(* Logix 5000 project; controller CarbonScout_MK6 vendor 1 type 14 code 154 rev 32.11; software revision 32.00; part 14 of 17 *)
(* tags used below, declared in another part *)
   i : DINT;
   Index : DINT;
   LocalSampleTank : DINT;
   LOnlineNumber : DINT;
   ManualRunning : BOOL;
   ONS : BOOL[32];
   TimeRemainingCal : TimeRemainingCal;
   AI_LIT_02 : P_AIn;   // Carbon Scout Cone Level Transmitter
   CS_DINTParams : DINT[100];
   CS_REALParams : REAL[80];   // CS REAL Parameters
   CS_ResultStore : CS_Results[20,20];   // Sample Result Historical
   CS_Seq : GEK_Sequence;
   CS_Tank : CS_TankParams[20];
   CS_Timer : TIMER[80];
   Reg_Cal : REAL[10];   // working calculation variables
   Reg_Calsum : REAL[10];   // running sum of calc variables
   Reg_DINTparams : DINT[8];   // Dint and bools for calcs
   Reg_InX : REAL[30];   // X input for calcs
   Reg_InY : REAL[30];   // Y input for pairs
   Reg_Model : REAL[4];   // Calculated model output and site model
   Reg_Out : REAL[14];   // Output of calculation
   TimeAndDate : DINT[7];
   Valve_XV_15 : P_ValveSO;   // Bottme wash vavle
(* SeqProgram, continued *)

ROUTINE DataShift   (* ladder *)
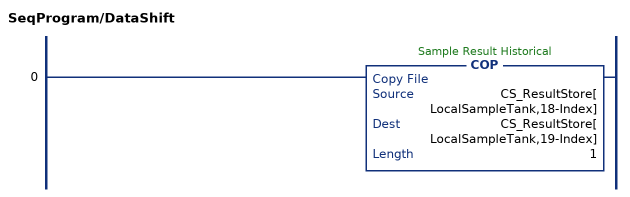
   0: COP(CS_ResultStore[LocalSampleTank,18-Index],CS_ResultStore[LocalSampleTank,19-Index],1);
END_ROUTINE

ROUTINE MainRoutine   (* ladder *)
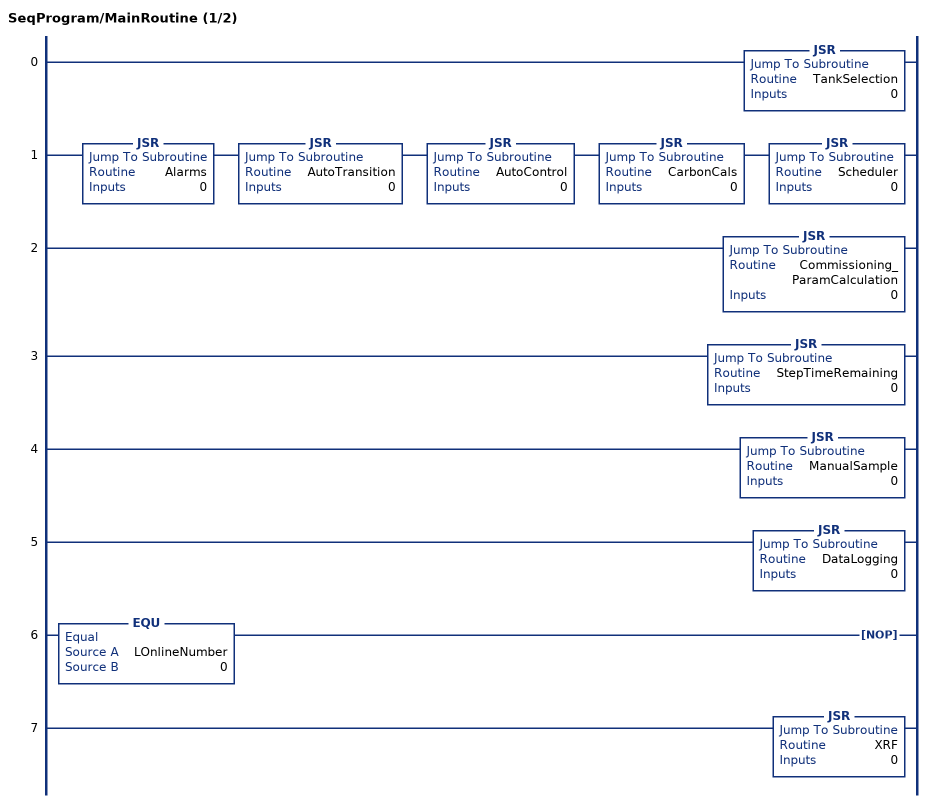
   0: JSR(TankSelection,0);
   1: JSR(Alarms,0)JSR(AutoTransition,0)JSR(AutoControl,0)JSR(CarbonCals,0)JSR(Scheduler,0);
   2: JSR(Commissioning_ParamCalculation,0);
   3: JSR(StepTimeRemaining,0);
   4: JSR(ManualSample,0);
   5: JSR(DataLogging,0);
   6: EQU(LOnlineNumber,0)NOP();
   7: JSR(XRF,0);
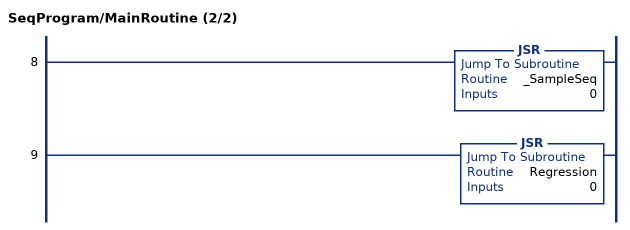
   8: JSR(_SampleSeq,0);
   9: JSR(Regression,0);
END_ROUTINE

ROUTINE ManualSample   (* ladder *)
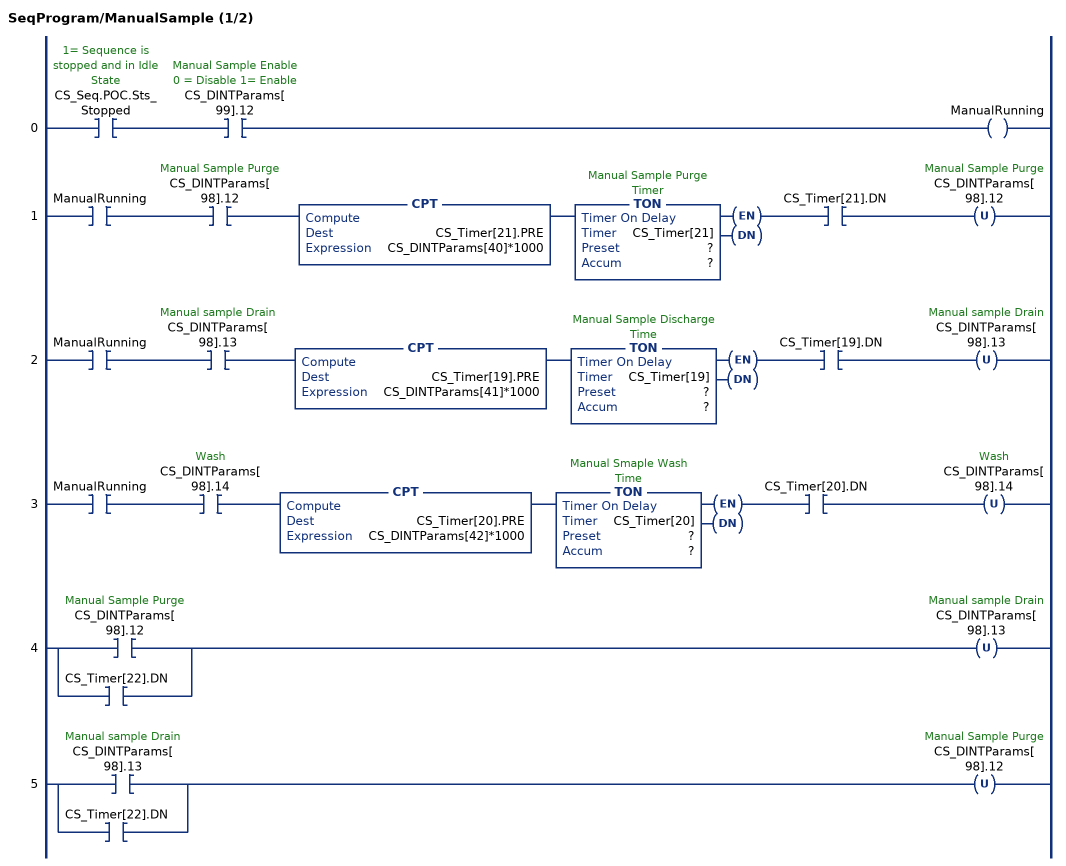
   0: XIC(CS_Seq.POC.Sts_Stopped)XIC(CS_DINTParams[99].12)OTE(ManualRunning);
   1: XIC(ManualRunning)XIC(CS_DINTParams[98].12)CPT(CS_Timer[21].PRE,CS_DINTParams[40]*1000)TON(CS_Timer[21],?,?)XIC(CS_Timer[21].DN)OTU(CS_DINTParams[98].12);
   2: XIC(ManualRunning)XIC(CS_DINTParams[98].13)CPT(CS_Timer[19].PRE,CS_DINTParams[41]*1000)TON(CS_Timer[19],?,?)XIC(CS_Timer[19].DN)OTU(CS_DINTParams[98].13);
   3: XIC(ManualRunning)XIC(CS_DINTParams[98].14)CPT(CS_Timer[20].PRE,CS_DINTParams[42]*1000)TON(CS_Timer[20],?,?)XIC(CS_Timer[20].DN)OTU(CS_DINTParams[98].14);
   4: [XIC(CS_DINTParams[98].12) ,XIC(CS_Timer[22].DN) ]OTU(CS_DINTParams[98].13);
   5: [XIC(CS_DINTParams[98].13) ,XIC(CS_Timer[22].DN) ]OTU(CS_DINTParams[98].12);
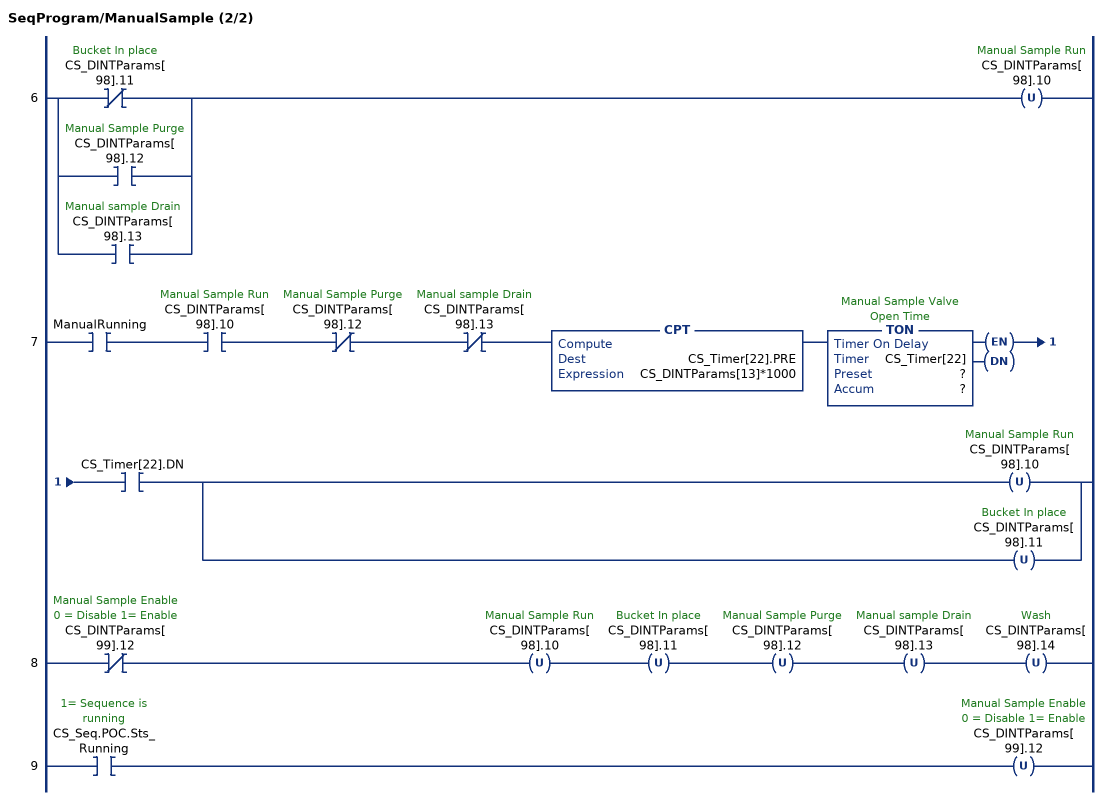
   6: [XIO(CS_DINTParams[98].11) ,XIC(CS_DINTParams[98].12) ,XIC(CS_DINTParams[98].13) ]OTU(CS_DINTParams[98].10);
   7: XIC(ManualRunning)XIC(CS_DINTParams[98].10)XIO(CS_DINTParams[98].12)XIO(CS_DINTParams[98].13)CPT(CS_Timer[22].PRE,CS_DINTParams[13]*1000)TON(CS_Timer[22],?,?)XIC(CS_Timer[22].DN)[OTU(CS_DINTParams[98].10) ,OTU(CS_DINTParams[98].11) ];
   8: XIO(CS_DINTParams[99].12)OTU(CS_DINTParams[98].10)OTU(CS_DINTParams[98].11)OTU(CS_DINTParams[98].12)OTU(CS_DINTParams[98].13)OTU(CS_DINTParams[98].14);
   9: XIC(CS_Seq.POC.Sts_Running)OTU(CS_DINTParams[99].12);
END_ROUTINE

ROUTINE Regression   (* ladder *)
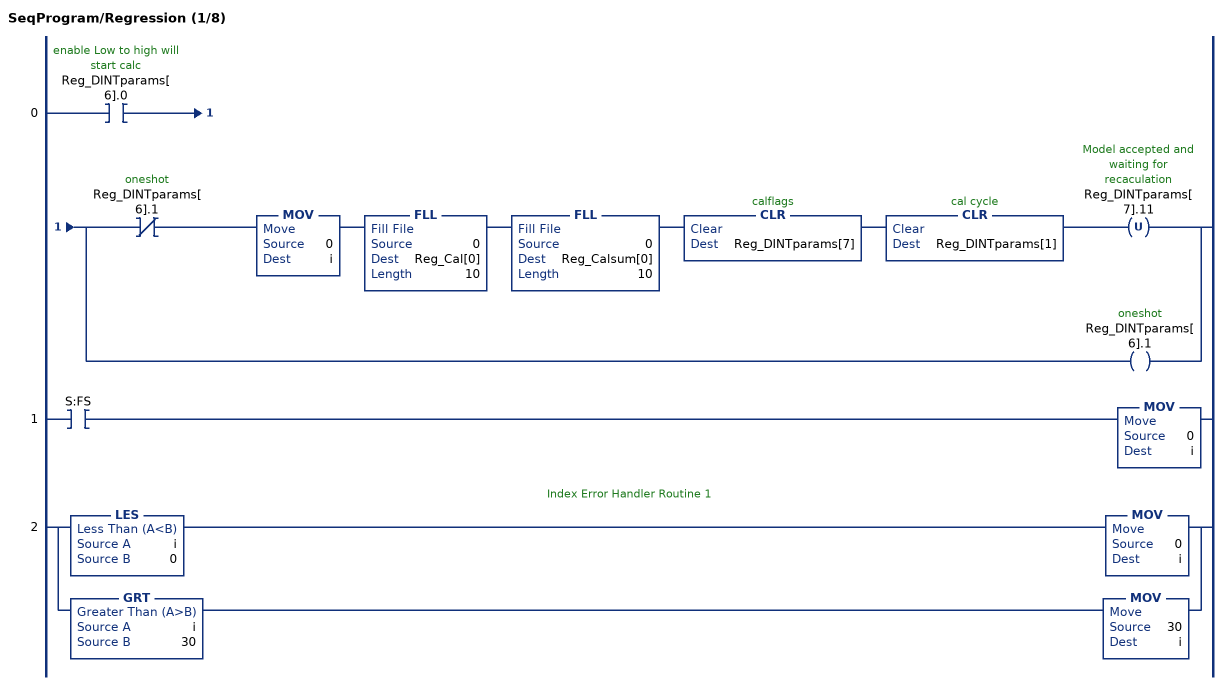
   0: XIC(Reg_DINTparams[6].0)[XIO(Reg_DINTparams[6].1) MOV(0,i) FLL(0,Reg_Cal[0],10) FLL(0,Reg_Calsum[0],10) CLR(Reg_DINTparams[7]) CLR(Reg_DINTparams[1]) OTU(Reg_DINTparams[7].11) ,OTE(Reg_DINTparams[6].1) ];
   1: XIC(S:FS)MOV(0,i);
   // Index Error Handler Routine 1
   2: [LES(i,0) MOV(0,i) ,GRT(i,30) MOV(30,i) ];
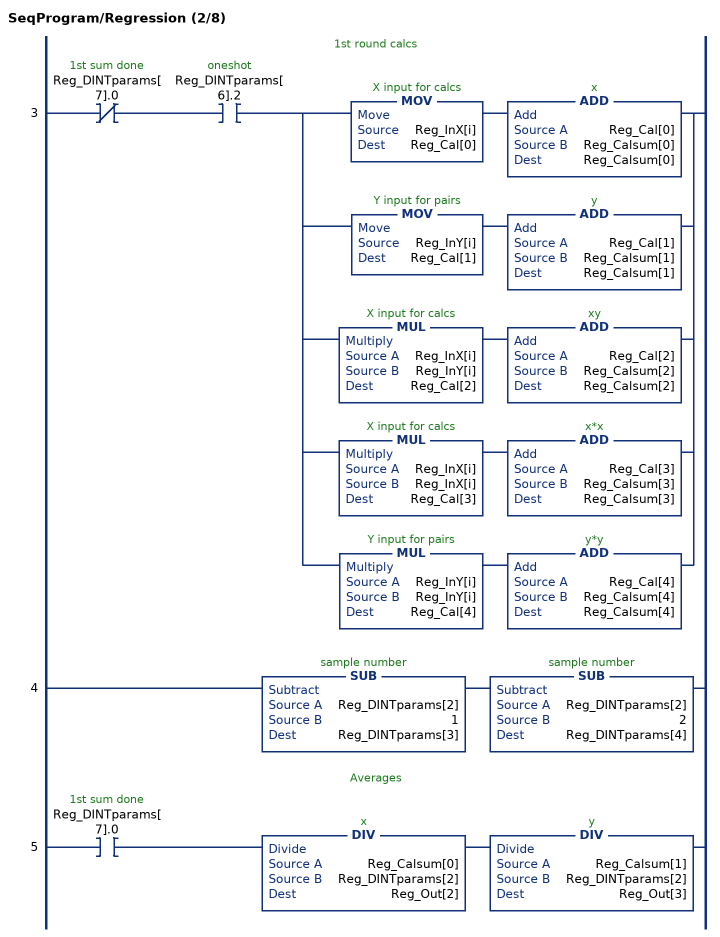
   // 1st round calcs
   3: XIO(Reg_DINTparams[7].0)XIC(Reg_DINTparams[6].2)[MOV(Reg_InX[i],Reg_Cal[0]) ADD(Reg_Cal[0],Reg_Calsum[0],Reg_Calsum[0]) ,MOV(Reg_InY[i],Reg_Cal[1]) ADD(Reg_Cal[1],Reg_Calsum[1],Reg_Calsum[1]) ,MUL(Reg_InX[i],Reg_InY[i],Reg_Cal[2]) ADD(Reg_Cal[2],Reg_Calsum[2],Reg_Calsum[2]) ,MUL(Reg_InX[i],Reg_InX[i],Reg_Cal[3]) ADD(Reg_Cal[3],Reg_Calsum[3],Reg_Calsum[3]) ,MUL(Reg_InY[i],Reg_InY[i],Reg_Cal[4]) ADD(Reg_Cal[4],Reg_Calsum[4],Reg_Calsum[4]) ];
   4: SUB(Reg_DINTparams[2],1,Reg_DINTparams[3])SUB(Reg_DINTparams[2],2,Reg_DINTparams[4]);
   // Averages
   5: XIC(Reg_DINTparams[7].0)DIV(Reg_Calsum[0],Reg_DINTparams[2],Reg_Out[2])DIV(Reg_Calsum[1],Reg_DINTparams[2],Reg_Out[3]);
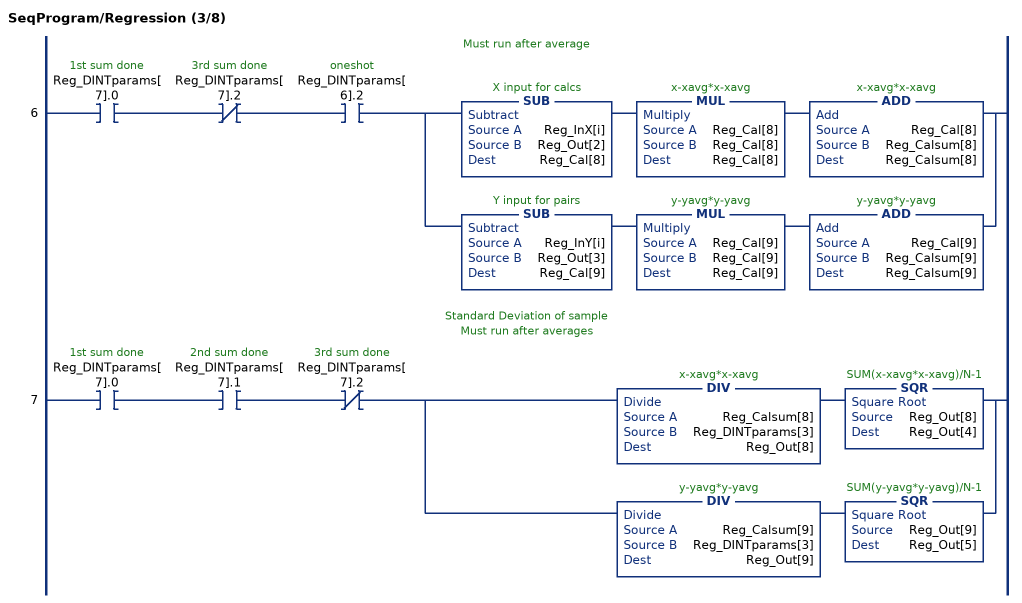
   // Must run after average
   6: XIC(Reg_DINTparams[7].0)XIO(Reg_DINTparams[7].2)XIC(Reg_DINTparams[6].2)[SUB(Reg_InX[i],Reg_Out[2],Reg_Cal[8]) MUL(Reg_Cal[8],Reg_Cal[8],Reg_Cal[8]) ADD(Reg_Cal[8],Reg_Calsum[8],Reg_Calsum[8]) ,SUB(Reg_InY[i],Reg_Out[3],Reg_Cal[9]) MUL(Reg_Cal[9],Reg_Cal[9],Reg_Cal[9]) ADD(Reg_Cal[9],Reg_Calsum[9],Reg_Calsum[9]) ];
   // Standard Deviation of sample
   // Must run after averages
   7: XIC(Reg_DINTparams[7].0)XIC(Reg_DINTparams[7].1)XIO(Reg_DINTparams[7].2)[DIV(Reg_Calsum[8],Reg_DINTparams[3],Reg_Out[8]) SQR(Reg_Out[8],Reg_Out[4]) ,DIV(Reg_Calsum[9],Reg_DINTparams[3],Reg_Out[9]) SQR(Reg_Out[9],Reg_Out[5]) ];
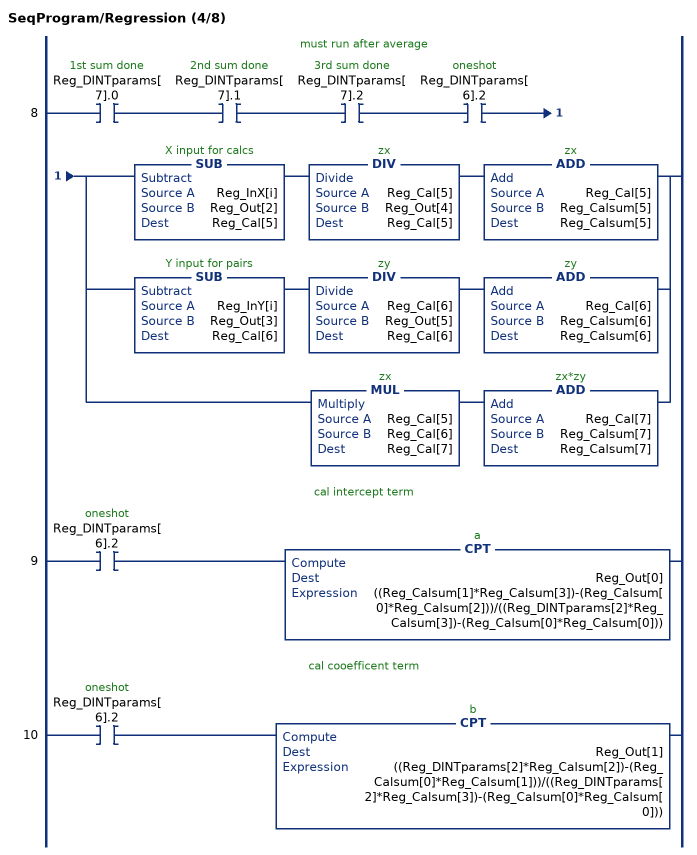
   // must run after average
   8: XIC(Reg_DINTparams[7].0)XIC(Reg_DINTparams[7].1)XIC(Reg_DINTparams[7].2)XIC(Reg_DINTparams[6].2)[SUB(Reg_InX[i],Reg_Out[2],Reg_Cal[5]) DIV(Reg_Cal[5],Reg_Out[4],Reg_Cal[5]) ADD(Reg_Cal[5],Reg_Calsum[5],Reg_Calsum[5]) ,SUB(Reg_InY[i],Reg_Out[3],Reg_Cal[6]) DIV(Reg_Cal[6],Reg_Out[5],Reg_Cal[6]) ADD(Reg_Cal[6],Reg_Calsum[6],Reg_Calsum[6]) ,MUL(Reg_Cal[5],Reg_Cal[6],Reg_Cal[7]) ADD(Reg_Cal[7],Reg_Calsum[7],Reg_Calsum[7]) ];
   // cal intercept term
   9: XIC(Reg_DINTparams[6].2)CPT(Reg_Out[0],((Reg_Calsum[1]*Reg_Calsum[3])-(Reg_Calsum[0]*Reg_Calsum[2]))/((Reg_DINTparams[2]*Reg_Calsum[3])-(Reg_Calsum[0]*Reg_Calsum[0])));
   // cal cooefficent term
   10: XIC(Reg_DINTparams[6].2)CPT(Reg_Out[1],((Reg_DINTparams[2]*Reg_Calsum[2])-(Reg_Calsum[0]*Reg_Calsum[1]))/((Reg_DINTparams[2]*Reg_Calsum[3])-(Reg_Calsum[0]*Reg_Calsum[0])));
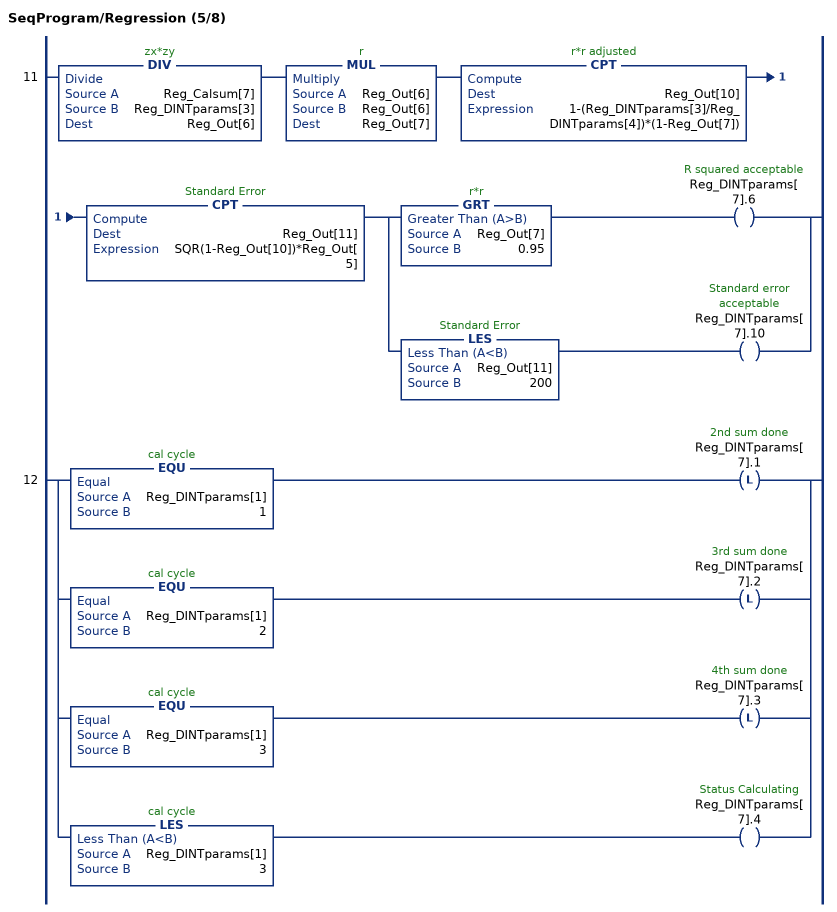
   11: DIV(Reg_Calsum[7],Reg_DINTparams[3],Reg_Out[6])MUL(Reg_Out[6],Reg_Out[6],Reg_Out[7])CPT(Reg_Out[10],1-(Reg_DINTparams[3]/Reg_DINTparams[4])*(1-Reg_Out[7]))CPT(Reg_Out[11],SQR(1-Reg_Out[10])*Reg_Out[5])[GRT(Reg_Out[7],0.95) OTE(Reg_DINTparams[7].6) ,LES(Reg_Out[11],200) OTE(Reg_DINTparams[7].10) ];
   12: [EQU(Reg_DINTparams[1],1) OTL(Reg_DINTparams[7].1) ,EQU(Reg_DINTparams[1],2) OTL(Reg_DINTparams[7].2) ,EQU(Reg_DINTparams[1],3) OTL(Reg_DINTparams[7].3) ,LES(Reg_DINTparams[1],3) OTE(Reg_DINTparams[7].4) ];
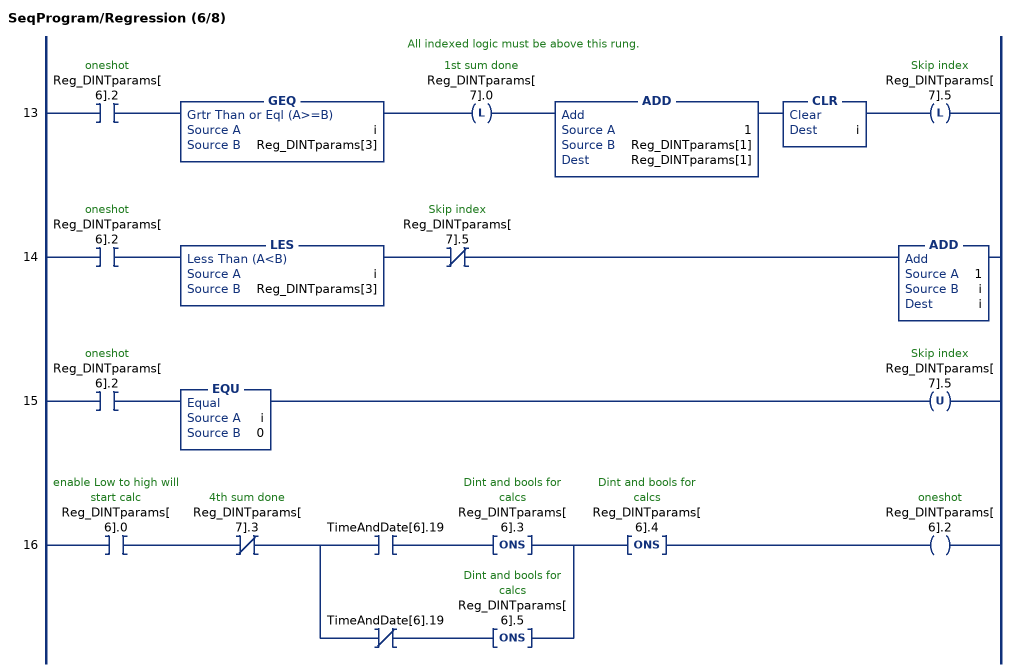
   // All indexed logic must be above this rung.
   13: XIC(Reg_DINTparams[6].2)GEQ(i,Reg_DINTparams[3])OTL(Reg_DINTparams[7].0)ADD(1,Reg_DINTparams[1],Reg_DINTparams[1])CLR(i)OTL(Reg_DINTparams[7].5);
   14: XIC(Reg_DINTparams[6].2)LES(i,Reg_DINTparams[3])XIO(Reg_DINTparams[7].5)ADD(1,i,i);
   15: XIC(Reg_DINTparams[6].2)EQU(i,0)OTU(Reg_DINTparams[7].5);
   16: XIC(Reg_DINTparams[6].0)XIO(Reg_DINTparams[7].3)[XIC(TimeAndDate[6].19) ONS(Reg_DINTparams[6].3) ,XIO(TimeAndDate[6].19) ONS(Reg_DINTparams[6].5) ]ONS(Reg_DINTparams[6].4)OTE(Reg_DINTparams[6].2);
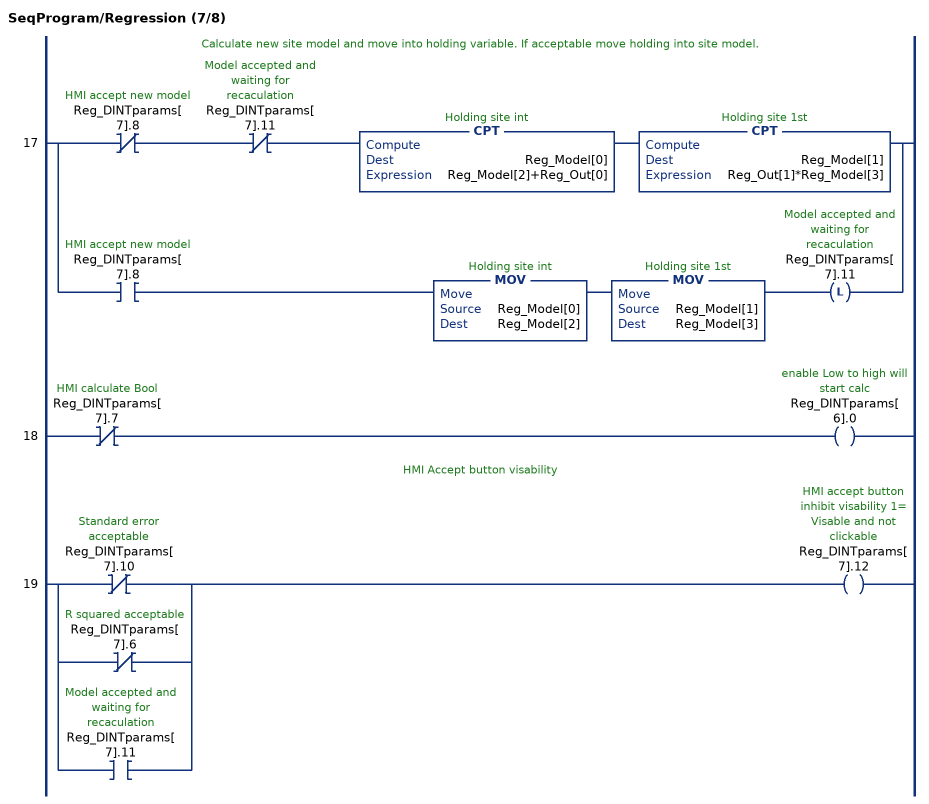
   // Calculate new site model and move into holding variable. If acceptable move holding into site model.
   17: [XIO(Reg_DINTparams[7].8) XIO(Reg_DINTparams[7].11) CPT(Reg_Model[0],Reg_Model[2]+Reg_Out[0]) CPT(Reg_Model[1],Reg_Out[1]*Reg_Model[3]) ,XIC(Reg_DINTparams[7].8) MOV(Reg_Model[0],Reg_Model[2]) MOV(Reg_Model[1],Reg_Model[3]) OTL(Reg_DINTparams[7].11) ];
   18: XIO(Reg_DINTparams[7].7)OTE(Reg_DINTparams[6].0);
   // HMI Accept button visability
   19: [XIO(Reg_DINTparams[7].10) ,XIO(Reg_DINTparams[7].6) ,XIC(Reg_DINTparams[7].11) ]OTE(Reg_DINTparams[7].12);
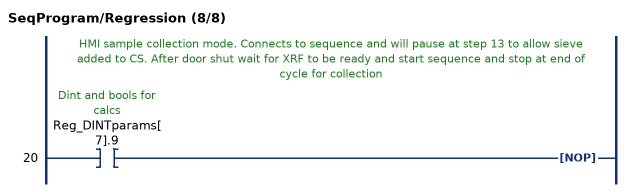
   // HMI sample collection mode. Connects to sequence and will pause at step 13 to allow sieve added to CS. After door shut wait for XRF to be ready and start sequence and stop at end of cycle for collection
   20: XIC(Reg_DINTparams[7].9)NOP();
END_ROUTINE

ROUTINE Scheduler   (* ladder *)
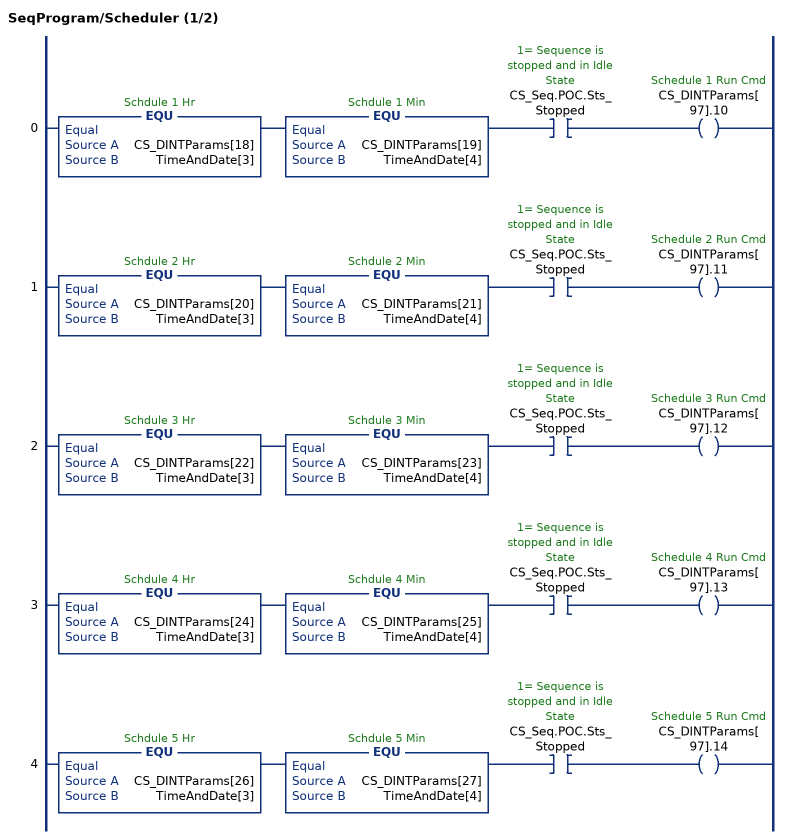
   0: EQU(CS_DINTParams[18],TimeAndDate[3])EQU(CS_DINTParams[19],TimeAndDate[4])XIC(CS_Seq.POC.Sts_Stopped)OTE(CS_DINTParams[97].10);
   1: EQU(CS_DINTParams[20],TimeAndDate[3])EQU(CS_DINTParams[21],TimeAndDate[4])XIC(CS_Seq.POC.Sts_Stopped)OTE(CS_DINTParams[97].11);
   2: EQU(CS_DINTParams[22],TimeAndDate[3])EQU(CS_DINTParams[23],TimeAndDate[4])XIC(CS_Seq.POC.Sts_Stopped)OTE(CS_DINTParams[97].12);
   3: EQU(CS_DINTParams[24],TimeAndDate[3])EQU(CS_DINTParams[25],TimeAndDate[4])XIC(CS_Seq.POC.Sts_Stopped)OTE(CS_DINTParams[97].13);
   4: EQU(CS_DINTParams[26],TimeAndDate[3])EQU(CS_DINTParams[27],TimeAndDate[4])XIC(CS_Seq.POC.Sts_Stopped)OTE(CS_DINTParams[97].14);
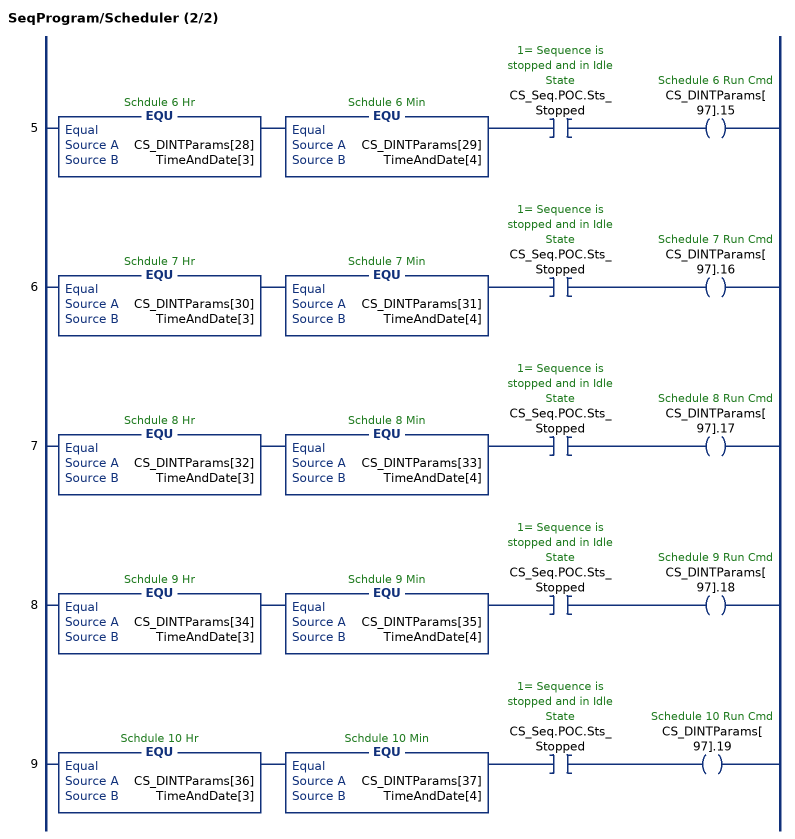
   5: EQU(CS_DINTParams[28],TimeAndDate[3])EQU(CS_DINTParams[29],TimeAndDate[4])XIC(CS_Seq.POC.Sts_Stopped)OTE(CS_DINTParams[97].15);
   6: EQU(CS_DINTParams[30],TimeAndDate[3])EQU(CS_DINTParams[31],TimeAndDate[4])XIC(CS_Seq.POC.Sts_Stopped)OTE(CS_DINTParams[97].16);
   7: EQU(CS_DINTParams[32],TimeAndDate[3])EQU(CS_DINTParams[33],TimeAndDate[4])XIC(CS_Seq.POC.Sts_Stopped)OTE(CS_DINTParams[97].17);
   8: EQU(CS_DINTParams[34],TimeAndDate[3])EQU(CS_DINTParams[35],TimeAndDate[4])XIC(CS_Seq.POC.Sts_Stopped)OTE(CS_DINTParams[97].18);
   9: EQU(CS_DINTParams[36],TimeAndDate[3])EQU(CS_DINTParams[37],TimeAndDate[4])XIC(CS_Seq.POC.Sts_Stopped)OTE(CS_DINTParams[97].19);
END_ROUTINE

ROUTINE StepTimeRemaining   (* ladder *)
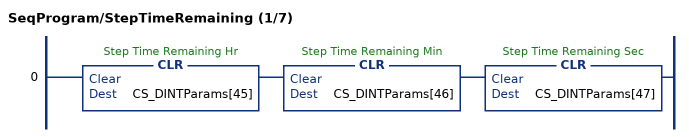
   0: CLR(CS_DINTParams[45])CLR(CS_DINTParams[46])CLR(CS_DINTParams[47]);
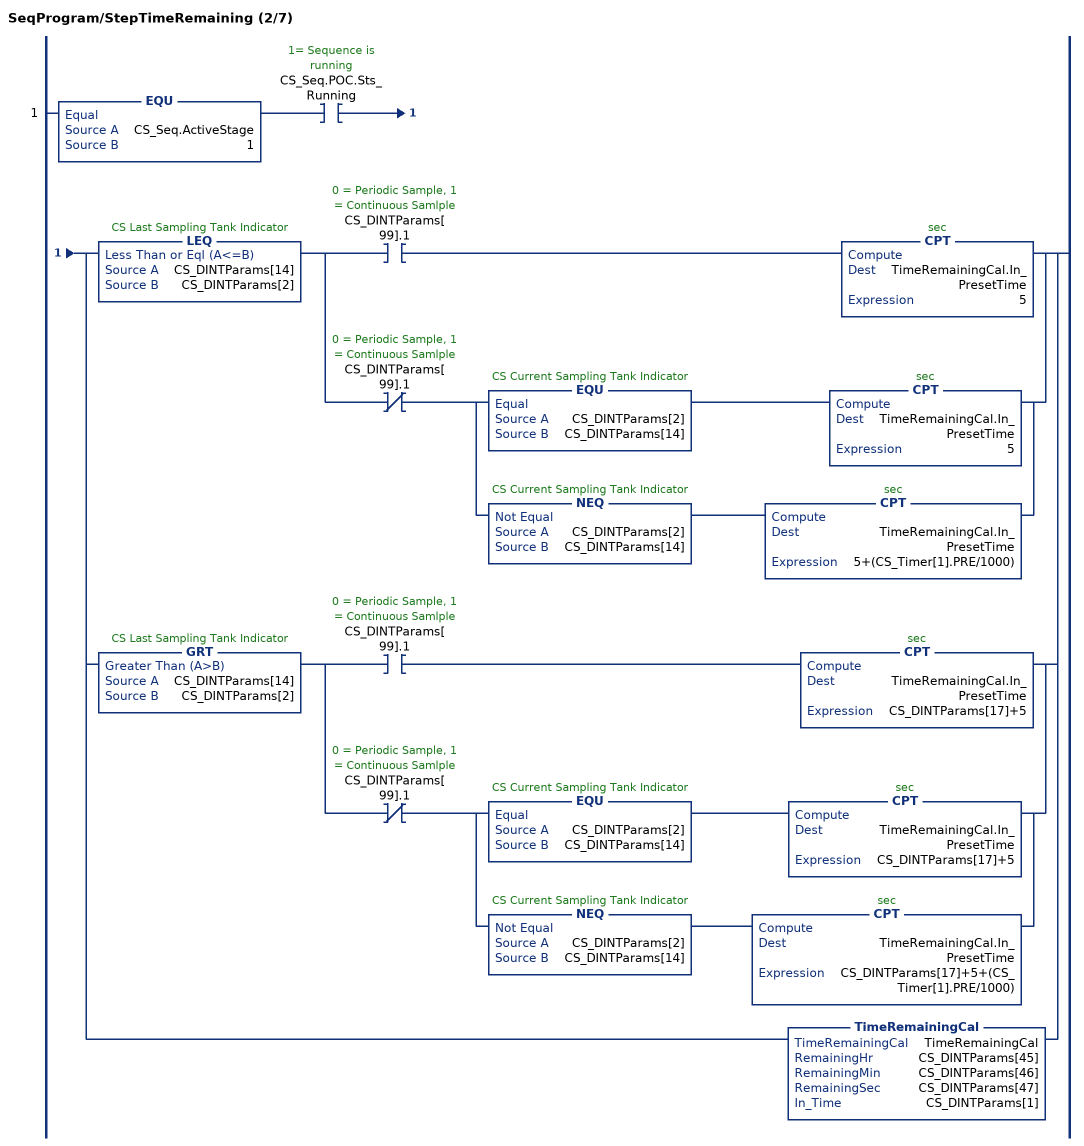
   1: EQU(CS_Seq.ActiveStage,1)XIC(CS_Seq.POC.Sts_Running)[[LEQ(CS_DINTParams[14],CS_DINTParams[2]) [XIC(CS_DINTParams[99].1) CPT(TimeRemainingCal.In_PresetTime,5) ,XIO(CS_DINTParams[99].1) [EQU(CS_DINTParams[2],CS_DINTParams[14]) CPT(TimeRemainingCal.In_PresetTime,5) ,NEQ(CS_DINTParams[2],CS_DINTParams[14]) CPT(TimeRemainingCal.In_PresetTime,5+(CS_Timer[1].PRE/1000)) ] ] ,GRT(CS_DINTParams[14],CS_DINTParams[2]) [XIC(CS_DINTParams[99].1) CPT(TimeRemainingCal.In_PresetTime,CS_DINTParams[17]+5) ,XIO(CS_DINTParams[99].1) [EQU(CS_DINTParams[2],CS_DINTParams[14]) CPT(TimeRemainingCal.In_PresetTime,CS_DINTParams[17]+5) ,NEQ(CS_DINTParams[2],CS_DINTParams[14]) CPT(TimeRemainingCal.In_PresetTime,CS_DINTParams[17]+5+(CS_Timer[1].PRE/1000)) ] ] ] ,TimeRemainingCal(TimeRemainingCal,CS_DINTParams[45],CS_DINTParams[46],CS_DINTParams[47],CS_DINTParams[1]) ];
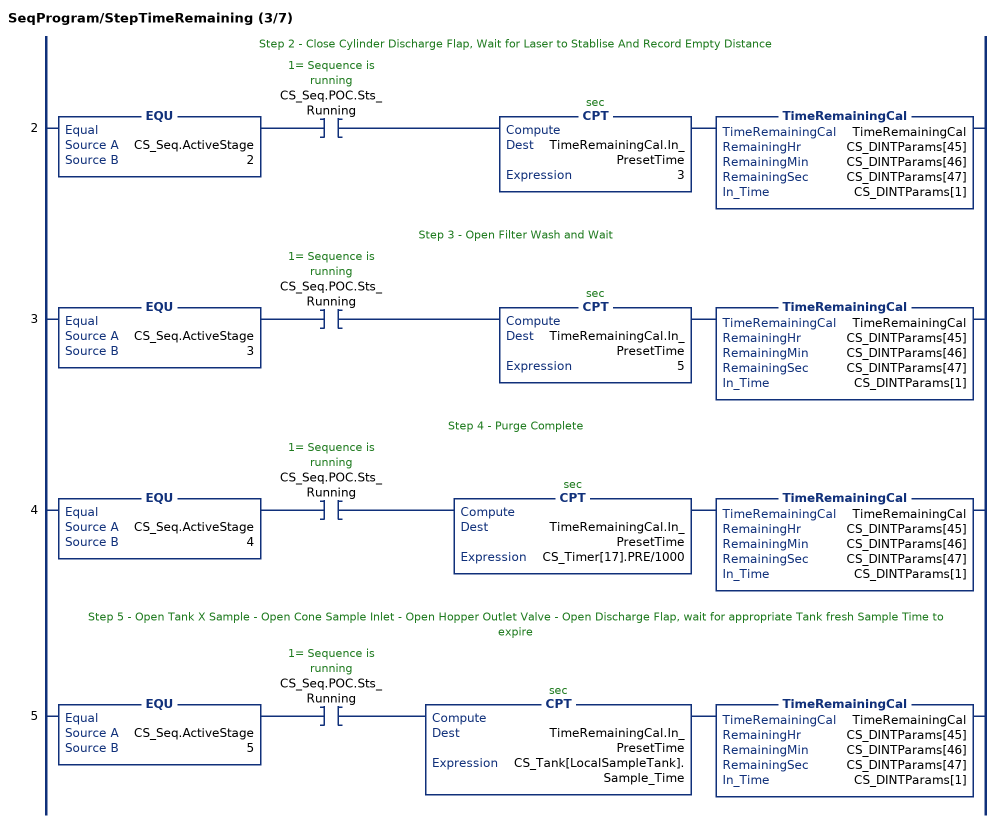
   // Step 2 - Close Cylinder Discharge Flap, Wait for Laser to Stablise And Record Empty Distance
   2: EQU(CS_Seq.ActiveStage,2)XIC(CS_Seq.POC.Sts_Running)CPT(TimeRemainingCal.In_PresetTime,3)TimeRemainingCal(TimeRemainingCal,CS_DINTParams[45],CS_DINTParams[46],CS_DINTParams[47],CS_DINTParams[1]);
   // Step 3 - Open Filter Wash and Wait
   3: EQU(CS_Seq.ActiveStage,3)XIC(CS_Seq.POC.Sts_Running)CPT(TimeRemainingCal.In_PresetTime,5)TimeRemainingCal(TimeRemainingCal,CS_DINTParams[45],CS_DINTParams[46],CS_DINTParams[47],CS_DINTParams[1]);
   // Step 4 - Purge Complete
   4: EQU(CS_Seq.ActiveStage,4)XIC(CS_Seq.POC.Sts_Running)CPT(TimeRemainingCal.In_PresetTime,CS_Timer[17].PRE/1000)TimeRemainingCal(TimeRemainingCal,CS_DINTParams[45],CS_DINTParams[46],CS_DINTParams[47],CS_DINTParams[1]);
   // Step 5 - Open Tank X Sample - Open Cone Sample Inlet - Open Hopper Outlet Valve - Open Discharge Flap, wait for appropriate Tank fresh Sample Time to expire
   5: EQU(CS_Seq.ActiveStage,5)XIC(CS_Seq.POC.Sts_Running)CPT(TimeRemainingCal.In_PresetTime,CS_Tank[LocalSampleTank].Sample_Time)TimeRemainingCal(TimeRemainingCal,CS_DINTParams[45],CS_DINTParams[46],CS_DINTParams[47],CS_DINTParams[1]);
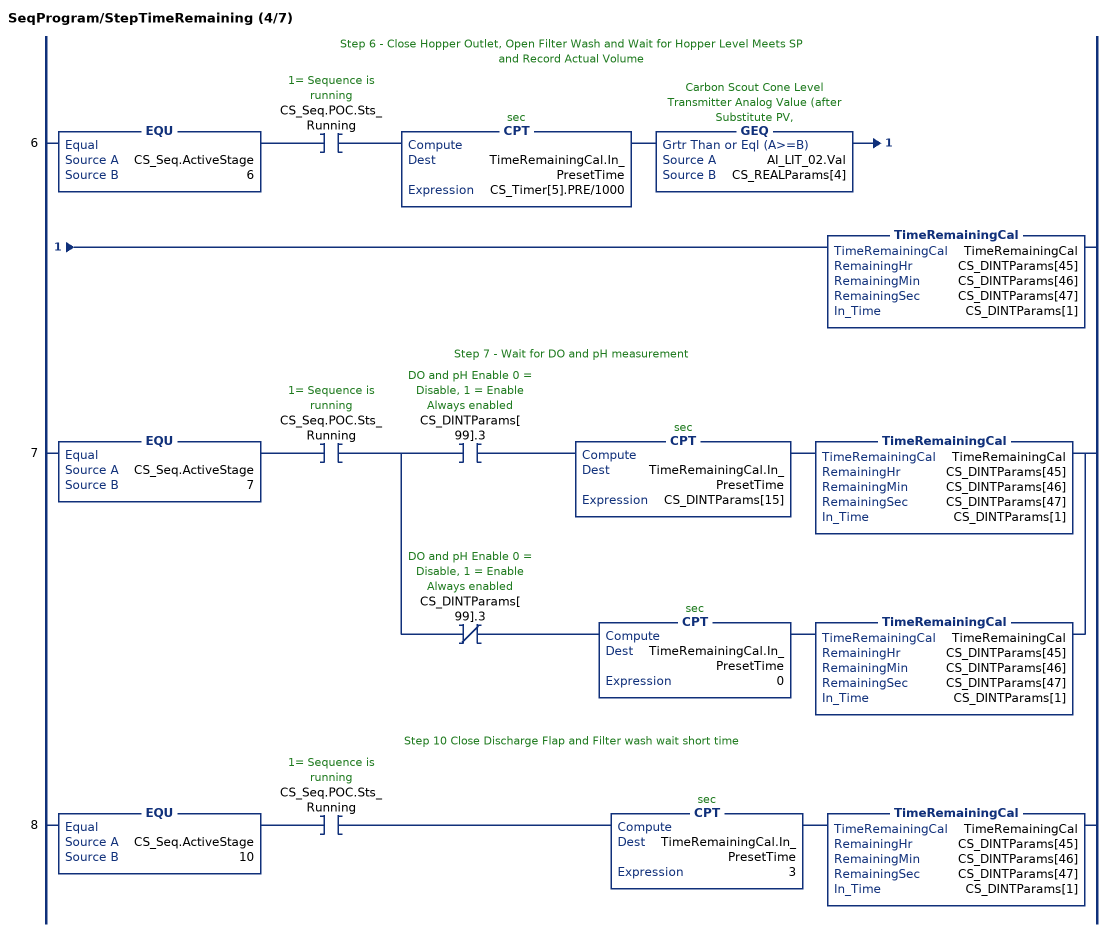
   // Step 6 - Close Hopper Outlet, Open Filter Wash and Wait for Hopper Level Meets SP
   // and Record Actual Volume
   6: EQU(CS_Seq.ActiveStage,6)XIC(CS_Seq.POC.Sts_Running)CPT(TimeRemainingCal.In_PresetTime,CS_Timer[5].PRE/1000)GEQ(AI_LIT_02.Val,CS_REALParams[4])TimeRemainingCal(TimeRemainingCal,CS_DINTParams[45],CS_DINTParams[46],CS_DINTParams[47],CS_DINTParams[1]);
   // Step 7 - Wait for DO and pH measurement
   7: EQU(CS_Seq.ActiveStage,7)XIC(CS_Seq.POC.Sts_Running)[XIC(CS_DINTParams[99].3) CPT(TimeRemainingCal.In_PresetTime,CS_DINTParams[15]) TimeRemainingCal(TimeRemainingCal,CS_DINTParams[45],CS_DINTParams[46],CS_DINTParams[47],CS_DINTParams[1]) ,XIO(CS_DINTParams[99].3) CPT(TimeRemainingCal.In_PresetTime,0) TimeRemainingCal(TimeRemainingCal,CS_DINTParams[45],CS_DINTParams[46],CS_DINTParams[47],CS_DINTParams[1]) ];
   // Step 10 Close Discharge Flap and Filter wash wait short time
   8: EQU(CS_Seq.ActiveStage,10)XIC(CS_Seq.POC.Sts_Running)CPT(TimeRemainingCal.In_PresetTime,3)TimeRemainingCal(TimeRemainingCal,CS_DINTParams[45],CS_DINTParams[46],CS_DINTParams[47],CS_DINTParams[1]);
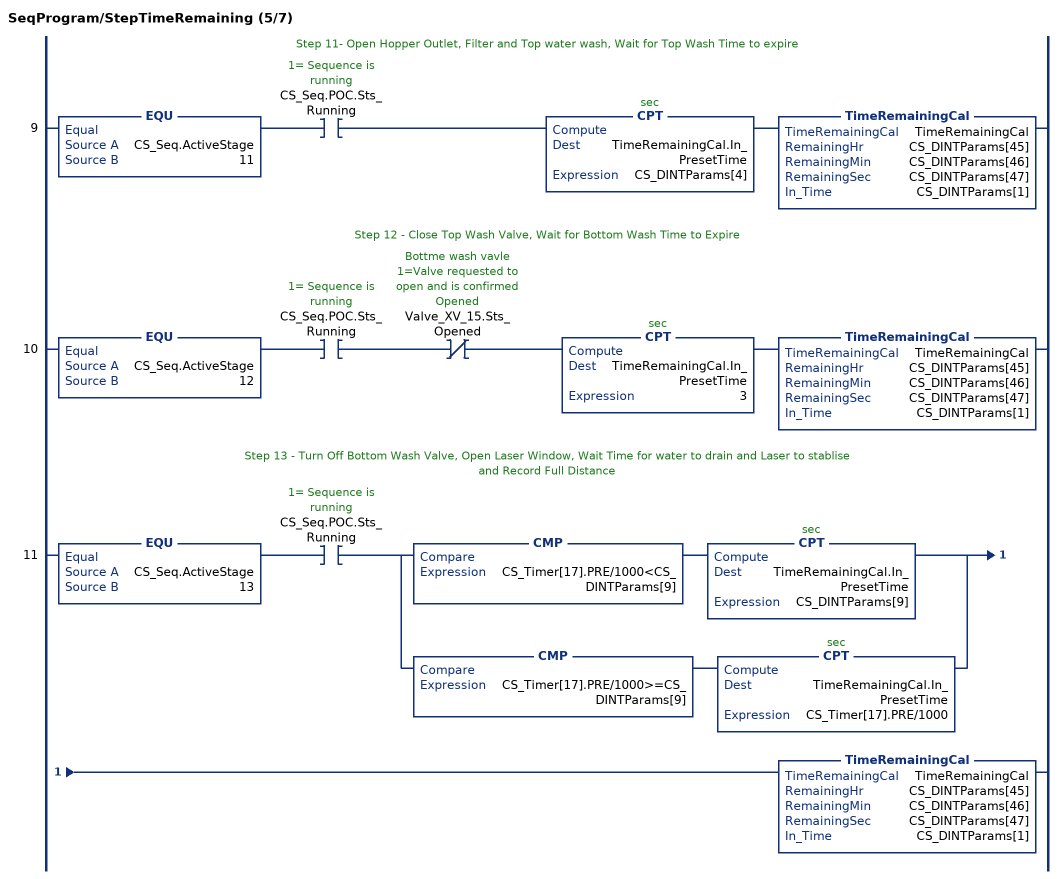
   // Step 11- Open Hopper Outlet, Filter and Top water wash, Wait for Top Wash Time to expire
   9: EQU(CS_Seq.ActiveStage,11)XIC(CS_Seq.POC.Sts_Running)CPT(TimeRemainingCal.In_PresetTime,CS_DINTParams[4])TimeRemainingCal(TimeRemainingCal,CS_DINTParams[45],CS_DINTParams[46],CS_DINTParams[47],CS_DINTParams[1]);
   // Step 12 - Close Top Wash Valve, Wait for Bottom Wash Time to Expire
   10: EQU(CS_Seq.ActiveStage,12)XIC(CS_Seq.POC.Sts_Running)XIO(Valve_XV_15.Sts_Opened)CPT(TimeRemainingCal.In_PresetTime,3)TimeRemainingCal(TimeRemainingCal,CS_DINTParams[45],CS_DINTParams[46],CS_DINTParams[47],CS_DINTParams[1]);
   // Step 13 - Turn Off Bottom Wash Valve, Open Laser Window, Wait Time for water to drain and Laser to stablise
   // and Record Full Distance
   11: EQU(CS_Seq.ActiveStage,13)XIC(CS_Seq.POC.Sts_Running)[CMP(CS_Timer[17].PRE/1000<CS_DINTParams[9]) CPT(TimeRemainingCal.In_PresetTime,CS_DINTParams[9]) ,CMP(CS_Timer[17].PRE/1000>=CS_DINTParams[9]) CPT(TimeRemainingCal.In_PresetTime,CS_Timer[17].PRE/1000) ]TimeRemainingCal(TimeRemainingCal,CS_DINTParams[45],CS_DINTParams[46],CS_DINTParams[47],CS_DINTParams[1]);
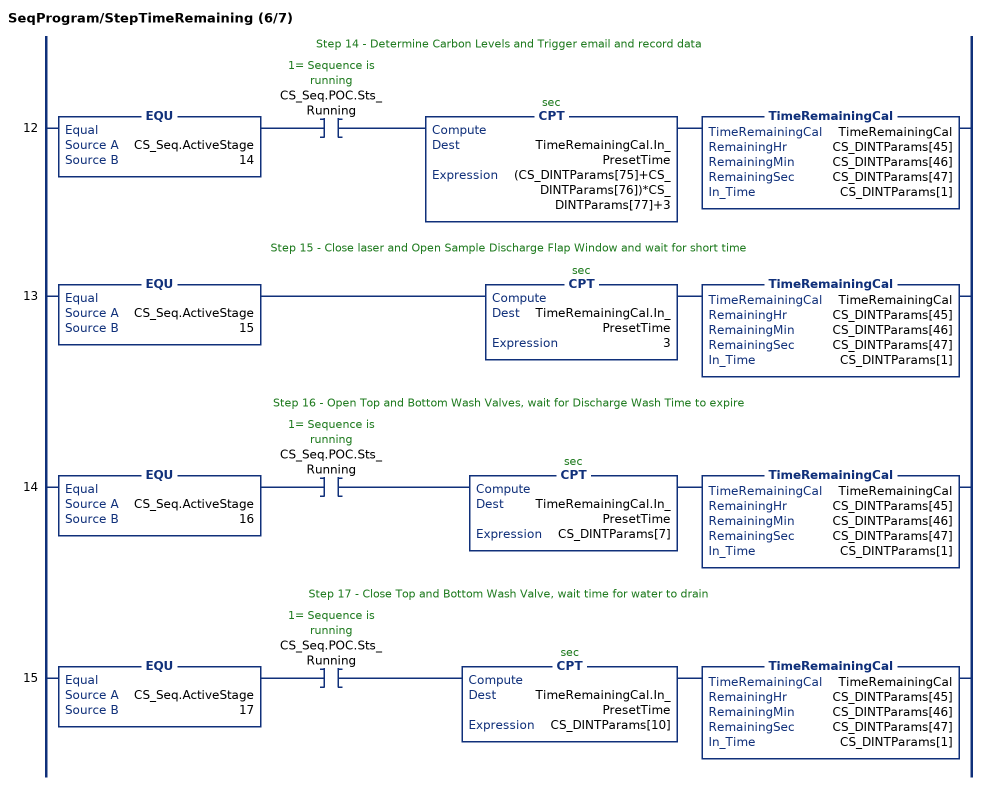
   // Step 14 - Determine Carbon Levels and Trigger email and record data
   12: EQU(CS_Seq.ActiveStage,14)XIC(CS_Seq.POC.Sts_Running)CPT(TimeRemainingCal.In_PresetTime,(CS_DINTParams[75]+CS_DINTParams[76])*CS_DINTParams[77]+3)TimeRemainingCal(TimeRemainingCal,CS_DINTParams[45],CS_DINTParams[46],CS_DINTParams[47],CS_DINTParams[1]);
   // Step 15 - Close laser and Open Sample Discharge Flap Window and wait for short time
   13: EQU(CS_Seq.ActiveStage,15)CPT(TimeRemainingCal.In_PresetTime,3)TimeRemainingCal(TimeRemainingCal,CS_DINTParams[45],CS_DINTParams[46],CS_DINTParams[47],CS_DINTParams[1]);
   // Step 16 - Open Top and Bottom Wash Valves, wait for Discharge Wash Time to expire
   14: EQU(CS_Seq.ActiveStage,16)XIC(CS_Seq.POC.Sts_Running)CPT(TimeRemainingCal.In_PresetTime,CS_DINTParams[7])TimeRemainingCal(TimeRemainingCal,CS_DINTParams[45],CS_DINTParams[46],CS_DINTParams[47],CS_DINTParams[1]);
   // Step 17 - Close Top and Bottom Wash Valve, wait time for water to drain
   15: EQU(CS_Seq.ActiveStage,17)XIC(CS_Seq.POC.Sts_Running)CPT(TimeRemainingCal.In_PresetTime,CS_DINTParams[10])TimeRemainingCal(TimeRemainingCal,CS_DINTParams[45],CS_DINTParams[46],CS_DINTParams[47],CS_DINTParams[1]);
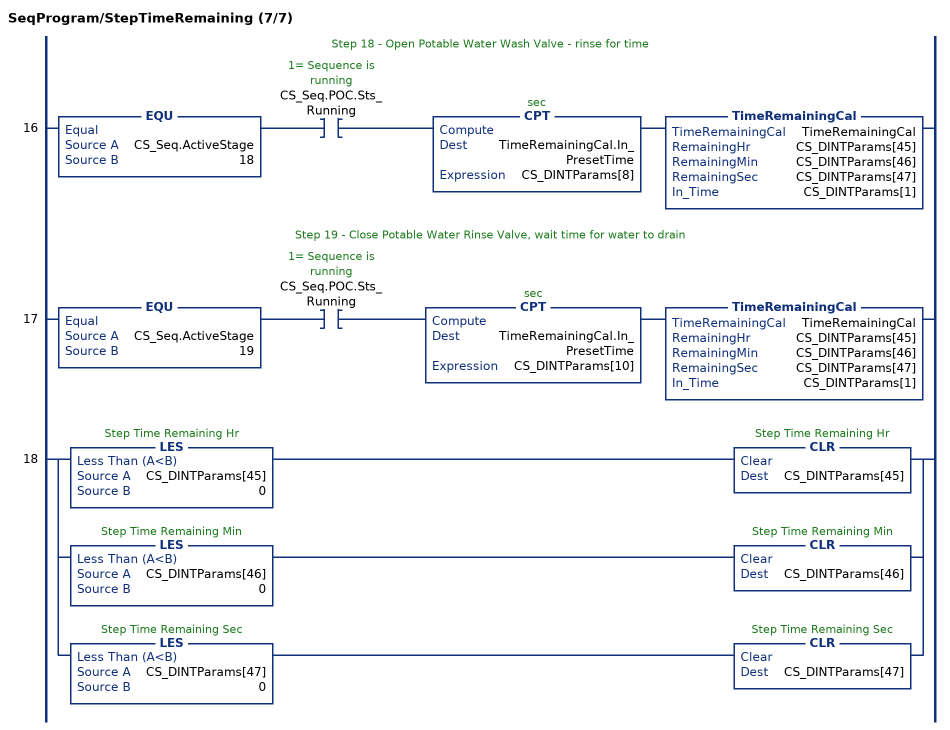
   // Step 18 - Open Potable Water Wash Valve - rinse for time
   16: EQU(CS_Seq.ActiveStage,18)XIC(CS_Seq.POC.Sts_Running)CPT(TimeRemainingCal.In_PresetTime,CS_DINTParams[8])TimeRemainingCal(TimeRemainingCal,CS_DINTParams[45],CS_DINTParams[46],CS_DINTParams[47],CS_DINTParams[1]);
   // Step 19 - Close Potable Water Rinse Valve, wait time for water to drain
   17: EQU(CS_Seq.ActiveStage,19)XIC(CS_Seq.POC.Sts_Running)CPT(TimeRemainingCal.In_PresetTime,CS_DINTParams[10])TimeRemainingCal(TimeRemainingCal,CS_DINTParams[45],CS_DINTParams[46],CS_DINTParams[47],CS_DINTParams[1]);
   18: [LES(CS_DINTParams[45],0) CLR(CS_DINTParams[45]) ,LES(CS_DINTParams[46],0) CLR(CS_DINTParams[46]) ,LES(CS_DINTParams[47],0) CLR(CS_DINTParams[47]) ];
END_ROUTINE
